(* PLC project Synergy Logic Function Blocks, OpenPLC Synergy Logic Function Blocks Library 1.0, author Synergy Logic *)
(* stored: creationDateTime 2021-11-11T02:33:11, modificationDateTime 2021-11-11T02:33:11 *)

(* Initialize SL Modules and return the number of initialized modules on SUCCESS. If SUCCESS is zero, an error has occurred, or there aren't any modules on the bus *)
FUNCTION_BLOCK SLM_INIT
  VAR_INPUT
    INIT : BOOL;
  END_VAR
  VAR_OUTPUT
    SUCCESS : BOOL;
  END_VAR

            SUCCESS := 0;
          
END_FUNCTION_BLOCK

(* UNITS: 1 = C/Low Burnout, 2 = C/High Burnout, 3 = F/Low Burnout, 3 = F/High Burnout CHANNELS: 0 = J, 1 = K, 2 = E, 3 = R, 4 = T, 5 = B, 6 = N, 7 = C *)
FUNCTION_BLOCK SLM_04THM_CONFIG
  VAR_INPUT
    SLOT : SINT;
    UNITS : SINT;
    CH1_RANGE : SINT;
    CH2_RANGE : SINT;
    CH3_RANGE : SINT;
    CH4_RANGE : SINT;
  END_VAR
  VAR_OUTPUT
    SUCCESS : BOOL;
  END_VAR

            SUCCESS := 0;
          
END_FUNCTION_BLOCK

(* Set all 8 channel outputs on discrete modules. *)
FUNCTION_BLOCK SLM_DISCRETE_OUT_8
  VAR_INPUT
    SLOT : SINT;
    O1 : BOOL;
    O2 : BOOL;
    O3 : BOOL;
    O4 : BOOL;
    O5 : BOOL;
    O6 : BOOL;
    O7 : BOOL;
    O8 : BOOL;
  END_VAR
  VAR
    DUMMY : SINT;
  END_VAR

            DUMMY := SLOT;
          
END_FUNCTION_BLOCK

(* Set all 15 channel outputs on discrete modules. *)
FUNCTION_BLOCK SLM_DISCRETE_OUT_15
  VAR_INPUT
    SLOT : SINT;
    O1 : BOOL;
    O2 : BOOL;
    O3 : BOOL;
    O4 : BOOL;
    O5 : BOOL;
    O6 : BOOL;
    O7 : BOOL;
    O8 : BOOL;
    O9 : BOOL;
    O10 : BOOL;
    O11 : BOOL;
    O12 : BOOL;
    O13 : BOOL;
    O14 : BOOL;
    O15 : BOOL;
  END_VAR
  VAR
    DUMMY : SINT;
  END_VAR

            DUMMY := SLOT;
          
END_FUNCTION_BLOCK

(* Set all 16 channel outputs on discrete modules. *)
FUNCTION_BLOCK SLM_DISCRETE_OUT_16
  VAR_INPUT
    SLOT : SINT;
    O1 : BOOL;
    O2 : BOOL;
    O3 : BOOL;
    O4 : BOOL;
    O5 : BOOL;
    O6 : BOOL;
    O7 : BOOL;
    O8 : BOOL;
    O9 : BOOL;
    O10 : BOOL;
    O11 : BOOL;
    O12 : BOOL;
    O13 : BOOL;
    O14 : BOOL;
    O15 : BOOL;
    O16 : BOOL;
  END_VAR
  VAR
    DUMMY : SINT;
  END_VAR

            DUMMY := SLOT;
          
END_FUNCTION_BLOCK

(* Get all 8 channel inputs on discrete modules. *)
FUNCTION_BLOCK SLM_DISCRETE_IN_8
  VAR_INPUT
    SLOT : SINT;
  END_VAR
  VAR_OUTPUT
    I1 : BOOL;
    I2 : BOOL;
    I3 : BOOL;
    I4 : BOOL;
    I5 : BOOL;
    I6 : BOOL;
    I7 : BOOL;
    I8 : BOOL;
  END_VAR

            I1 := 0;
          
END_FUNCTION_BLOCK

(* Get all 16 channel inputs on discrete modules. *)
FUNCTION_BLOCK SLM_DISCRETE_IN_16
  VAR_INPUT
    SLOT : SINT;
  END_VAR
  VAR_OUTPUT
    I1 : BOOL;
    I2 : BOOL;
    I3 : BOOL;
    I4 : BOOL;
    I5 : BOOL;
    I6 : BOOL;
    I7 : BOOL;
    I8 : BOOL;
    I9 : BOOL;
    I10 : BOOL;
    I11 : BOOL;
    I12 : BOOL;
    I13 : BOOL;
    I14 : BOOL;
    I15 : BOOL;
    I16 : BOOL;
  END_VAR

            I1 := 0;
          
END_FUNCTION_BLOCK

(* Get all 4 channel inputs on analog modules *)
FUNCTION_BLOCK SLM_ANALOG_IN_4
  VAR_INPUT
    SLOT : SINT;
  END_VAR
  VAR_OUTPUT
    I1 : UINT;
    I2 : UINT;
    I3 : UINT;
    I4 : UINT;
  END_VAR
  VAR
    DUMMY : SINT;
  END_VAR

            DUMMY := SLOT;
          
END_FUNCTION_BLOCK

(* Get all 4 channel inputs on analog modules *)
FUNCTION_BLOCK SLM_ANALOG_IN_8
  VAR_INPUT
    SLOT : SINT;
  END_VAR
  VAR_OUTPUT
    I1 : UINT;
    I2 : UINT;
    I3 : UINT;
    I4 : UINT;
    I5 : UINT;
    I6 : UINT;
    I7 : UINT;
    I8 : UINT;
  END_VAR
  VAR
    DUMMY : SINT;
  END_VAR

            DUMMY := SLOT;
          
END_FUNCTION_BLOCK

(* Set all 4 channel outputs on analog modules *)
FUNCTION_BLOCK SLM_ANALOG_OUT_4
  VAR_INPUT
    SLOT : SINT;
    O1 : UINT;
    O2 : UINT;
    O3 : UINT;
    O4 : UINT;
  END_VAR
  VAR
    DUMMY : SINT;
  END_VAR

            DUMMY := SLOT;
          
END_FUNCTION_BLOCK

(* Set all 8 channel outputs on analog modules *)
FUNCTION_BLOCK SLM_ANALOG_OUT_8
  VAR_INPUT
    SLOT : SINT;
    O1 : UINT;
    O2 : UINT;
    O3 : UINT;
    O4 : UINT;
    O5 : UINT;
    O6 : UINT;
    O7 : UINT;
    O8 : UINT;
  END_VAR
  VAR
    DUMMY : SINT;
  END_VAR

            DUMMY := SLOT;
          
END_FUNCTION_BLOCK

(* Get all 4 channel inputs on temperature modules *)
FUNCTION_BLOCK SLM_TEMPERATURE_4
  VAR_INPUT
    SLOT : SINT;
  END_VAR
  VAR_OUTPUT
    I1 : REAL;
    I2 : REAL;
    I3 : REAL;
    I4 : REAL;
  END_VAR
  VAR
    DUMMY : SINT;
  END_VAR

            DUMMY := SLOT;
          
END_FUNCTION_BLOCK
